FUNCTION_BLOCK FB_DetectFlicker
// Detect if a booleean variable is flickering 

VAR_INPUT
	IN_VAR			: BOOL;						// Boolean input to analyze
	IN_Window		: TIME := T#5S;				// Time Window during which I check the number of value change
	IN_Count		: UINT;						// Maximum number of change for the tiume duration 

END_VAR
VAR_OUTPUT
	OUT_bFlicker		: BOOL;					// Value is considered as flickering
END_VAR
VAR
	COUNT 			: CTU ; 
	TON				: TON ; 
END_VAR

TON(IN:= TRUE , PT:= IN_Window ) ; 

IF COUNT.CV > IN_Count THEN 
	OUT_bFlicker := TRUE ; 
ELSIF COUNT.CV < IN_Count AND TON.Q THEN  
	OUT_bFlicker := FALSE ; 
END_IF	
	
COUNT(CU:= IN_VAR , PV:= 1000 , RESET:=TON.Q)  ; 

IF TON.Q THEN 
	TON(IN:= FALSE ) ; 
END_IF

END_FUNCTION_BLOCK

(* stored: Version 1.1.0.1, ProductVersion 3.1.4024.6
   POU FB_DetectFlicker: Id {dcd89db8-3f12-4281-a3ed-f6022f87649c}, SpecialFunc None *)
